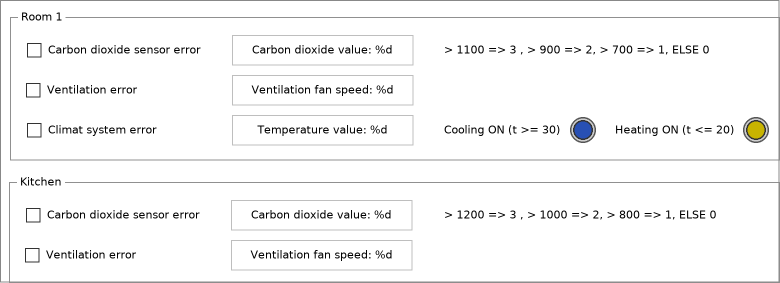
VISUALIZATION Visualization  // 780x283
    GroupBox (10,9 770x151), "Room 1"
        Checkbox (15,26 192x30), "Carbon dioxide sensor error", variable: MAIN.SmartHome.CarbonDioxideSensor_Room_1.ErrorSimulation
        Checkbox (14,66 193x30), "Ventilation error", variable: MAIN.SmartHome.Ventilation_Room_1.ErrorSimulation
        Checkbox (15,106 191x30), "Climat system error", variable: MAIN.SmartHome.ClimatSystem_Room_1.ErrorSimulation
        Textfield (222,26 181x30), "Carbon dioxide value: %d", text variable: MAIN.SmartHome.CarbonDioxideSensor_Room_1._CarbonDioxideLevel
            OnMouseClick: write the text variable via Default
        Textfield (222,66 181x30), "Ventilation fan speed: %d", text variable: MAIN.SmartHome.Ventilation_Room_1._Speed
        Textfield (222,106 181x30), "Temperature value: %d", text variable: MAIN.SmartHome.ClimatSystem_Room_1._Temperature
            OnMouseClick: write the text variable via Default
        Label (431,106 120x30), "Cooling ON (t >= 30)"
        Lamp1 (553,106 40x30), variable: MAIN.SmartHome.ClimatSystem_Room_1._IsCoolingOn, style: Lamp-Lamp1-Blue
        Label (602,106 123x30), "Heating ON (t <= 20)"
        Lamp1 (726,106 40x30), variable: MAIN.SmartHome.ClimatSystem_Room_1._IsHeatingOn, style: Lamp-Lamp1-Yellow
        Label (431,26 328x30), "> 1100 => 3 , > 900 => 2, > 700 => 1, ELSE 0"
    GroupBox (9,174 771x109), "Kitchen"
        Checkbox (15,26 192x30), "Carbon dioxide sensor error", variable: MAIN.SmartHome.CarbonDioxideSensor_Kitchen.ErrorSimulation
        Checkbox (14,66 193x30), "Ventilation error", variable: MAIN.SmartHome.Ventilation_Kitchen.ErrorSimulation
        Textfield (222,26 181x30), "Carbon dioxide value: %d", text variable: MAIN.SmartHome.CarbonDioxideSensor_Kitchen._CarbonDioxideLevel
            OnMouseClick: write the text variable via Default
        Textfield (222,66 181x30), "Ventilation fan speed: %d", text variable: MAIN.SmartHome.Ventilation_Kitchen._Speed
        Label (432,26 328x30), "> 1200 => 3 , > 1000 => 2, > 800 => 1, ELSE 0"
END_VISUALIZATION

(* stored: Version 1.1.0.1
   Visu Visualization: Id {11f42637-dedf-4be1-ac8e-44d1b5e64e90} *)
